PROGRAM MAIN
VAR
END_VAR

END_PROGRAM

(* stored: Version 1.1.0.1
   POU MAIN: Id {cd80c5e5-8640-472c-9c3b-079b376c8955} *)
